(* IEC 61131-3 sources: AceDryControl/Avfuktare/src/Application/Function_Blocks, 3 files *)

(* ---- AorB_2Values.iecst ---- *)
FUNCTION_BLOCK FB_TwoChannelSelect

    VAR_INPUT
        EnA   : BOOL;   // Enable för kanal A
        EnB   : BOOL;   // Enable för kanal B
        A_Val1 : REAL;  // Värde 1 för kanal A
        A_Val2 : REAL;  // Värde 2 för kanal A
        B_Val1 : REAL;  // Värde 1 för kanal B
        B_Val2 : REAL;  // Värde 2 för kanal B
    END_VAR

    VAR_OUTPUT
        OutVal1 : REAL; // Valt värde 1
        OutVal2 : REAL; // Valt värde 2
    END_VAR

    // Default
    OutVal1 := 0.0;
    OutVal2 := 0.0;

    // Prioritet: A först, annars B, annars default
    IF EnA THEN
        OutVal1 := A_Val1;
        OutVal2 := A_Val2;
    ELSIF EnB THEN
        OutVal1 := B_Val1;
        OutVal2 := B_Val2;
    ELSE
        // Ingen enable -> behåll default (0.0 / 0.0)
        OutVal1 := 0.0;
        OutVal2 := 0.0;
    END_IF;

END_FUNCTION_BLOCK

(* ---- IfAnyTrue3_1.iecst ---- *)
FUNCTION_BLOCK FB_AnyTrue3  {
    expandableGUI;
    safeStyle;
    width := 160;
  }
    VAR_INPUT
        In1 : BOOL;
        In2 : BOOL;
        In3 : BOOL;
    END_VAR

    VAR_OUTPUT
        Out : BOOL;
    END_VAR

    // Default
    Out := FALSE;

    // Om någon är TRUE -> Out TRUE
    IF In1 OR In2 OR In3 THEN
        Out := TRUE;
    END_IF;

END_FUNCTION_BLOCK

(* ---- OpModeSelector.iecst ---- *)
FUNCTION_BLOCK FB_ModeSelector  {
    altName := "ModeSelector";
    width := 180;
    instanceName;
    safeStyle;
    height := 78;
    minWidth := 0;
  }
	VAR_INPUT
	    OpMode : UINT;   // 0=Off, 1=Manual, 2=AutoRH, 3=AutoAH
	END_VAR

	VAR_OUTPUT
	    Off    : BOOL;
	    Manual    : BOOL;
	    AutoRH  : BOOL;
	    AutoAH : BOOL;
	END_VAR

	// Default
	Off    := FALSE;
	Manual     := FALSE;
	AutoRH  := FALSE;
	AutoAH := FALSE;

    CASE OpMode OF
        0: Off    := TRUE;
        1: Manual     := TRUE;
        2: AutoRH  := TRUE;
        3: AutoAH := TRUE;
    ELSE
        // fail-safe
        Off := TRUE;
    END_CASE;
END_FUNCTION_BLOCK
